PROGRAM MAIN
VAR

END_VAR

PRG_VLS_MOTION(); // So, run the program associated with coupler

END_PROGRAM

(* stored: Version 1.1.0.1, ProductVersion 3.1.4020.14
   POU MAIN: Id {e6fa2b58-86f6-4521-8196-c6010dfb509b}, SpecialFunc None *)
